// This file does not demonstrate the PLC BaseVista concept. It's used for PlcCommunication testing.
VAR_GLOBAL
	strDefaultString	: STRING;
	strLongString		: STRING(160);
	strShortString		: STRING(5);
	
	bolTest		: BOOL;
END_VAR

(* stored: Version 1.1.0.1, ProductVersion 3.1.0.19
   GVL Test: Id {a0e3f84f-fcc8-4f32-ace5-ed43414fb32e} *)
